{attribute 'GeneratedUsingTerminal: ELX4181-0000-0016'}
{attribute addProperty BoxType "ELX4181-0000-0016"}
{attribute addProperty Id "AO_OutputsAO_Output_Channel_BA7EBB7C2"}
{attribute addProperty CRC "701764233"}
{attribute addProperty Size "2"}
TYPE Ch_1_29D41289 :
STRUCT
	{attribute addProperty Name "AO_Outputs"}
	AO_Outputs  : AO_Output_Channel_BA7EBB7C;
END_STRUCT
END_TYPE

(* stored: Version 1.2.0.0, ProductVersion 3.1.4024.9
   DUT Ch_1_29D41289: Id {0b512e0f-e672-4913-a646-eecb80925b53} *)
